// TIA Portal V20 export
DATA_BLOCK "DB_BwLoaderExchange"   // DB101
{ S7_Optimized_Access := 'TRUE' }
// stored: MemoryReserve 100
   VAR
      Inputs : Struct
         LifeFlag : Int;
         JobDone : Bool;
         LockShuttle : Bool;
         DataSend : Int;
         DataReceive : Int;
         NoEmergencyStopAtBwLoader : Bool;
         SafetyDoorsClosedAtBwLoader : Bool;
         BwInErrorState : Int;
         UndrilledPartControl : Bool;
         DrilledPartControl : Bool;
         BackwallControl : Bool;
         BwLoaderInSafePos : Bool;
      END_STRUCT;
      Outputs : Struct
         LifeFlag : Int;
         LoaderRequest : Bool;
         LockShuttle : Bool;
         DataSend : Int;
         DataReceive : Int;
         NoEmergencyStopAtFemto : Bool;
         SafetyDoorsClosedAtFemto : Bool;
         FemtoInErrorState : Int;
         AutoMode : Bool;
         JogMode : Bool;
         GotoSafePos : Bool;
         Emptying : Bool;
         BW_CtrlInProgress : Bool;
      END_STRUCT;
   END_VAR
BEGIN
END_DATA_BLOCK
